// TwinCAT 3 PLC project Intecre_Events
// Title: Intecre.Events
// Company: Intecre Ltd
// Author: Mit Patel
// ProjectVersion: 0.1.1.2
// Description: V0.1.1.0 - Initial V0.1.1.1 - Create RPC Sink V0.1.1.2 - Separate Buffer and Sink Interfaces
// ProgramVersion: 3.1.4024.0
// libraries:
//   Intecre.Utilities, * (Intecre Ltd)
//   Tc2_EtherCAT, * (Beckhoff Automation GmbH)
//   Tc2_Standard, * (Beckhoff Automation GmbH)
//   Tc2_System, * (Beckhoff Automation GmbH)
//   Tc2_Utilities, * (Beckhoff Automation GmbH)
//   Tc3_JsonXml, * (Beckhoff Automation GmbH)
//   Intecre.File,newest,Intecre Ltd
// project tree:
//   Library/EventLogger/EventBuffers/ T_JsonEventBuffer.TcPOU (not stored)
//   Library/EventLogger/EventSinks/ T_RpcEventSink.TcPOU, FB_CsvFileEventSink.TcPOU
//   Library/EventLogger/Interfaces/ I_EventSink.TcIO, I_EventBuffer.TcIO, I_EventLogger.TcIO, I_Logger.TcIO (not stored), I_EventSeverityHandler.TcIO, I_EventSinkHandler.TcIO (not stored)
//   Library/Structs/ ST_EventMessageBuffer.TcDUT, ST_EventMessageBufferPool.TcDUT (not stored), ST_EventMessageParams.TcDUT (not stored), T_BufferString.TcDUT (not stored), T_MessageString.TcDUT
//   Library/EventLogger/Bases/ T_InstanceNameBase.TcPOU
//   Library/EventLogger/Functions/ F_GetLogSeverityFromTcEventSeverity.TcPOU
//   Library/EventLogger/ T_EventLogger.TcPOU, T_Logger.TcPOU (not stored)
//   Library/GVLs/ Events.TcGVL (not stored), EventsConfig.TcGVL
//   Library/Time/ FB_UnixTimestamp.TcPOU (not stored), I_TimeProvider.TcIO
//   Project Information/ F_GetCompany.TcPOU, F_GetTitle.TcPOU, F_GetVersion.TcPOU
//   Version/ Global_Version.TcGVL

// ---- Library/Structs/ST_EventMessageBuffer.TcDUT
{attribute 'pack_mode' := '0'}
TYPE ST_EventMessageBuffer :
STRUCT
 	bufferIndex : UINT := 0;
	availableForWriting : BOOL := TRUE;
  count : UINT := 0;
  timestampMs : ULINT;
  
  bufferSize : UDINT := EventsConfig.MAX_BUFFER_SIZE;
  dataSize : UDINT := 0;
END_STRUCT
END_TYPE

// ---- Library/Structs/T_MessageString.TcDUT
TYPE T_MessageString : STRING(EventsConfig.MAX_LOG_MESSAGE_SIZE); END_TYPE

// ---- Library/GVLs/EventsConfig.TcGVL
{attribute 'qualified_only'}
// Buffer Config
VAR_GLOBAL CONSTANT
  MAX_BUFFERS : UINT := 4;                    // Number of buffers.
  MAX_BUFFER_SIZE : UDINT := 65535;           // Max size in bytes of a buffer.
  CYCLE_BUFFERS : BOOL := TRUE;               // Overwrite buffers when all buffers are full.
  MAX_LOG_MESSAGE_SIZE : UINT := 512;         // Max length of log message.
  
  CSV_LOG_FILE_NAME : T_MaxString := 'logs';      // Name for CSV log files. Will have the date appended (e.g. logs_2024_05_26).
  CSV_LOG_FILE_PATH : T_MaxString := '/var/log/'; // The path for log files if using FB_CsvFileEventSink.
END_VAR

// Logs config
VAR_GLOBAL CONSTANT
  MAX_SINKS : UINT := 4; // Number of sinks.
END_VAR

// ---- Version/Global_Version.TcGVL
{attribute 'TcGenerated'}
{attribute 'no-analysis'}
{attribute 'linkalways'}
// This function has been automatically generated from the project information.
VAR_GLOBAL CONSTANT
	{attribute 'const_non_replaced'}
	stLibVersion_Intecre_Events : ST_LibVersion := (iMajor := 0, iMinor := 1, iBuild := 1, iRevision := 2, nFlags := 0, sVersion := '0.1.1.2');
END_VAR

// ---- Library/EventLogger/Interfaces/I_EventSink.TcIO
// Interface for consuming and exposing event logs for transmitting to an event receiver/ listener.
INTERFACE I_EventSink

// Adds an event to the sink for processing.
METHOD AddEvent
VAR_INPUT
  eventMessageParams : ST_EventMessageParams;
END_VAR
END_METHOD

// Gets events currently stored in the buffer and copies them to the resultString.
METHOD GetEvents : T_BufferString;
END_METHOD

// Initialises the sink including an I_TimeProvider for timestamping events.
METHOD Initialise
VAR_INPUT
	timeProvider : I_TimeProvider;
END_VAR
END_METHOD

END_INTERFACE

// ---- Library/EventLogger/Interfaces/I_EventBuffer.TcIO
// Interface for buffering event logs.
INTERFACE I_EventBuffer

// Adds an event to the buffer for later processing.
METHOD AddEvent
VAR_INPUT
  eventMessageParams : ST_EventMessageParams;
END_VAR
END_METHOD

// Gets events currently stored in the buffer and copies them to the resultString, returning the total length of bytes copied.
METHOD GetEvents : UDINT
VAR_INPUT
  resultString : REFERENCE TO T_BufferString;
END_VAR
END_METHOD

// Initialises the buffer including an I_TimeProvider for timestamping buffers and events.
METHOD Initialise
VAR_INPUT
	timeProvider : I_TimeProvider;
END_VAR
END_METHOD

END_INTERFACE

// ---- Library/EventLogger/Interfaces/I_EventLogger.TcIO
// Internal interface for general logging methods required by all loggers.
INTERFACE INTERNAL I_EventLogger

// Generic logging method.
METHOD INTERNAL LogEvent
VAR_IN_OUT CONSTANT
  message : T_MessageString; 
  sourceInstanceName : T_MaxString;
END_VAR

VAR_INPUT
  severity : TcEventSeverity;
END_VAR
END_METHOD

// Checks severity filters for whether the log message/ event should be logged.
METHOD INTERNAL ShouldLogEvent : BOOL
VAR_INPUT
  severity : TcEventSeverity;
END_VAR
END_METHOD

END_INTERFACE

// ---- Library/EventLogger/Interfaces/I_EventSeverityHandler.TcIO
// Interface for setting/ clearing local severity level.
INTERFACE I_EventSeverityHandler

// Clear the currently set local severity level.
METHOD ClearLocalSeverity
END_METHOD

// Get global severity level.
METHOD GetGlobalSeverity : TcEventSeverity
END_METHOD

// Get local severity level.
METHOD GetLocalSeverity : TcEventSeverity
END_METHOD

// Set a global severity level to filter logged events.
METHOD SetGlobalSeverity
VAR_INPUT
  severity : TcEventSeverity;
END_VAR
END_METHOD

// Set a local severity level to filter logged events. Ensure clear is called once local logging is complete.
METHOD SetLocalSeverity
VAR_INPUT
  severity : TcEventSeverity;
END_VAR
END_METHOD

END_INTERFACE

// ---- Library/Time/I_TimeProvider.TcIO
INTERFACE I_TimeProvider

PROPERTY TimestampMs : ULINT
GET
END_GET
END_PROPERTY

END_INTERFACE

// ---- Library/EventLogger/EventSinks/FB_CsvFileEventSink.TcPOU
// Event sink which writes log messages/ events to a CSV file. 
FUNCTION_BLOCK PUBLIC FB_CsvFileEventSink EXTENDS T_InstanceNameBase IMPLEMENTS I_EventSink
VAR
  isInitialised : BOOL := FALSE;
  
  csvFileWriter : T_CsvFileWriter;
  
  _timeProvider : I_TimeProvider := NULL;
  
  // Timeout timer to write messages in the T_CsvFileWriter's buffer after a timeout period.
  timeoutDuration : TIME := T#2S;         
  startTimer : BOOL := TRUE;
  timeoutTrigger : TON := (IN := startTimer, PT := timeoutDuration);
  
  task : T_Task;
  currentDateTime : T_MaxString;
  eventId : ULINT := 0;
END_VAR

VAR CONSTANT
  NULL : UDINT := 0;
END_VAR

// Adds an event to the sink for processing.
METHOD PUBLIC AddEvent
VAR_INPUT
  eventMessageParams : ST_EventMessageParams;
END_VAR
IF NOT isInitialised THEN
  F_LogWarning(CONCAT(InstanceName, ': Unable to AddEvent. Sink is uninitialised.'));
  RETURN;
END_IF

IF task.DateString <> currentDateTime THEN
  currentDateTime := task.DateString;
  csvFileWriter.SetFileParams(F_Concat3(EventsConfig.CSV_LOG_FILE_PATH, F_Concat3(EventsConfig.CSV_LOG_FILE_NAME, '_', currentDateTime), '.csv'), ASCI_COMMA);
END_IF

csvFileWriter.AddStringField(TO_STRING(eventId));
csvFileWriter.AddStringField(TO_STRING(_timeProvider.TimestampMs));
csvFileWriter.AddStringField(TO_STRING(eventMessageParams.Severity));
csvFileWriter.AddStringField(eventMessageParams.Source);
csvFileWriter.AddStringField(eventMessageParams.Message);

// Todo. Additional fields, unix timestamp, event id etc.

csvFileWriter.NewLine();
eventId := eventId + 1;
END_METHOD

METHOD PUBLIC CyclicLogic
IF NOT isInitialised THEN
  F_LogWarning(CONCAT(InstanceName, ': Unable to Execute. Sink is uninitialised.'));
  RETURN;
END_IF

csvFileWriter();

timeoutTrigger(IN := startTimer); // Restart timer on next cycle if triggered
IF timeoutTrigger.Q THEN
  timeoutTrigger(IN := FALSE);
  GetEvents();                    // Write data in the buffer.
END_IF
END_METHOD

// Gets events currently stored in the buffer and copies them to the resultString.
METHOD PUBLIC GetEvents : T_BufferString;
IF NOT isInitialised THEN
  F_LogWarning(CONCAT(InstanceName, ': Unable to GetEvents. Sink is uninitialised.'));
  RETURN;
END_IF

csvFileWriter.WriteToFile();
END_METHOD

// Initialises the buffer including an I_TimeProvider for timestamping buffers and events.
METHOD PUBLIC Initialise
VAR_INPUT
	timeProvider : I_TimeProvider;
END_VAR
_timeProvider := timeProvider;

IF _timeProvider = NULL THEN
  F_LogWarning(CONCAT(InstanceName, ': Unable to Initialise. _timeProvider is uninitialised.'));
  RETURN;
END_IF

isInitialised := TRUE;

currentDateTime := task.DateString;
csvFileWriter.SetFileOpenMode(TRUE);
csvFileWriter.SetFileParams(F_Concat3(EventsConfig.CSV_LOG_FILE_PATH, F_Concat3(EventsConfig.CSV_LOG_FILE_NAME, '_', currentDateTime), '.csv'), ASCI_COMMA);
END_METHOD

END_FUNCTION_BLOCK

// ---- Library/EventLogger/Bases/T_InstanceNameBase.TcPOU
{attribute 'reflection'} 
FUNCTION_BLOCK PUBLIC T_InstanceNameBase
VAR
  {attribute 'instance-path'} 
  {attribute 'noinit'} 
  name : T_MaxString;
  
  _instanceName : T_MaxString;
  isInstanceNameSet : BOOL := FALSE;
END_VAR

PROPERTY FINAL InstanceName : T_MaxString; // returns the fully scoped variable name
GET
IF NOT isInstanceNameSet THEN
   setInstanceName();
END_IF

InstanceName := _instanceName;
END_GET
END_PROPERTY

METHOD PRIVATE SetInstanceName
VAR
	charsToDeleteFromPath : INT;
END_VAR
//Remove Solution_Name
charsToDeleteFromPath := FIND(name, '.');
_instanceName := DELETE(name, charsToDeleteFromPath, 1);
//Remove ProjectName
charsToDeleteFromPath := FIND(_instanceName, '.');
//gives us just "FirstDeclaredPOU.etc.etc..." from above.
_instanceName := DELETE(_instanceName, charsToDeleteFromPath, 1);
END_METHOD

END_FUNCTION_BLOCK

// ---- Library/EventLogger/EventSinks/T_RpcEventSink.TcPOU
// Event sink which buffers log messages/ events ready for polling via RPC calls to 'GetEvents'; a method of the I_EventSink interface. 
FUNCTION_BLOCK PUBLIC T_RpcEventSink EXTENDS T_InstanceNameBase IMPLEMENTS I_EventSink
VAR
  jsonBuffer : T_JsonEventBuffer;
END_VAR

// Adds an event to the sink for processing.
METHOD PUBLIC AddEvent
VAR_INPUT
  eventMessageParams : ST_EventMessageParams;
END_VAR
jsonBuffer.AddEvent(eventMessageParams);
END_METHOD

// Gets events currently stored in the buffer and copies them to the resultString.
{attribute 'TcRpcEnable'}
METHOD PUBLIC GetEvents : T_BufferString;
jsonBuffer.GetEvents(GetEvents);
END_METHOD

// Initialises the buffer including an I_TimeProvider for timestamping buffers and events.
METHOD PUBLIC Initialise
VAR_INPUT
	timeProvider : I_TimeProvider;
END_VAR
jsonBuffer.Initialise(timeProvider);
END_METHOD

END_FUNCTION_BLOCK

// ---- Library/EventLogger/Functions/F_GetLogSeverityFromTcEventSeverity.TcPOU
// Conversion helper to convert from TcEventSeverity to Intecre.Utilities E_LogSeverity.
FUNCTION INTERNAL F_GetLogSeverityFromTcEventSeverity : E_LogSeverity
VAR_INPUT
  severity : TcEventSeverity;
END_VAR

CASE severity OF

  TcEventSeverity.Verbose   : F_GetLogSeverityFromTcEventSeverity := E_LogSeverity.Debug;
  TcEventSeverity.Info      : F_GetLogSeverityFromTcEventSeverity := E_Logseverity.Info;
  TcEventSeverity.Warning   : F_GetLogSeverityFromTcEventSeverity := E_Logseverity.Warning;
  TcEventSeverity.Error     : F_GetLogSeverityFromTcEventSeverity := E_Logseverity.Error;
  TcEventSeverity.Critical  : F_GetLogSeverityFromTcEventSeverity := E_Logseverity.Error;

END_CASE

END_FUNCTION

// ---- Library/EventLogger/T_EventLogger.TcPOU
// Internal logger which allows adding/ clearing sinks to be processed, in addition to receiving log events and forwarding them to sinks.
FUNCTION_BLOCK INTERNAL T_EventLogger EXTENDS T_InstanceNameBase IMPLEMENTS I_EventLogger, I_Logger, I_EventSinkHandler, I_EventSeverityHandler;
VAR
  eventSinks : ARRAY[1..EventsConfig.MAX_SINKS] OF I_EventSink;
  eventSinksCount : UINT := 0;
  
  globalSeverity : TcEventSeverity; // Global log filter.
  localSeverity : TcEventSeverity;
  useLocalSeverity : BOOL;
END_VAR

VAR CONSTANT
  NULL : UDINT := 0;
END_VAR

// Adds a sink to the sink handler and returns TRUE if successful.
METHOD PUBLIC AddSink : BOOL
VAR_INPUT
	sink	: I_EventSink;
END_VAR
IF eventSinksCount + 1 > EventsConfig.MAX_SINKS THEN
  F_LogWarning(CONCAT(InstanceName, ': Unable to add sink. Maximum number of event sinks reached'));
  RETURN;
END_IF

eventSinksCount := eventSinksCount + 1;
eventSinks[eventSinksCount] := sink;
AddSink := TRUE;
END_METHOD

// Clear the currently set local severity level.
METHOD PUBLIC ClearLocalSeverity
useLocalSeverity := FALSE;
END_METHOD

// Clears all sinks currently being handled by the sink handler.
METHOD PUBLIC ClearSinks
VAR
  iSink : UINT := 0;
END_VAR
IF eventSinksCount > 0 AND eventSinksCount <= EventsConfig.MAX_SINKS THEN
  FOR iSink := 1 TO eventSinksCount DO
    eventSinks[iSink] := NULL;
  END_FOR
END_IF

eventSinksCount := 0;
END_METHOD

// Get global severity level.
METHOD GetGlobalSeverity : TcEventSeverity
GetGlobalSeverity := globalSeverity;
END_METHOD

// Get local severity level.
METHOD GetLocalSeverity : TcEventSeverity
GetLocalSeverity := localSeverity;
END_METHOD

METHOD PUBLIC LogCritical
VAR_INPUT
  message : T_MessageString; 
END_VAR

VAR
  localInstanceName : T_MaxString;
END_VAR
localInstanceName := InstanceName;
LogEvent(message := message, sourceInstanceName := localInstanceName, severity := TcEventSeverity.Critical);
END_METHOD

METHOD PUBLIC LogError
VAR_INPUT
  message : T_MessageString; 
END_VAR

VAR
  localInstanceName : T_MaxString;
END_VAR
localInstanceName := InstanceName;
LogEvent(message := message, sourceInstanceName := localInstanceName, severity := TcEventSeverity.Error);
END_METHOD

METHOD INTERNAL LogEvent
VAR_IN_OUT CONSTANT
  message : T_MessageString; 
  sourceInstanceName : T_MaxString;
END_VAR

VAR_INPUT
  severity : TcEventSeverity;
END_VAR

VAR
  iSink : UINT := 0;
  adsLogSeverity : E_LogSeverity;
  eventMessageParams : ST_EventMessageParams;
END_VAR
IF NOT ShouldLogEvent(severity) THEN
  RETURN;
END_IF

eventMessageParams.Message := message;
eventMessageParams.Severity := severity;
eventMessageParams.Source := sourceInstanceName;

IF eventSinksCount > 0 AND eventSinksCount <= EventsConfig.MAX_SINKS THEN
  FOR iSink := 1 TO eventSinksCount DO
    IF eventSinks[iSink] <> NULL THEN
      eventSinks[iSink].AddEvent(eventMessageParams);
    ELSE
      F_LogWarning(CONCAT(InstanceName, ': Unable to LogEvent. Sink is uninitialised.'));
    END_IF
  END_FOR
END_IF

adsLogSeverity := F_GetLogSeverityFromTcEventSeverity(severity);
F_Logger(
  LogSeverity := adsLogSeverity,
  Message := F_Concat3(sourceInstanceName, ': ', message)
);
END_METHOD

METHOD PUBLIC LogInfo
VAR_INPUT
  message : T_MessageString; 
END_VAR

VAR
  localInstanceName : T_MaxString;
END_VAR
localInstanceName := InstanceName;
LogEvent(message := message, sourceInstanceName := localInstanceName, severity := TcEventSeverity.Info);
END_METHOD

METHOD PUBLIC LogVerbose
VAR_INPUT
  message : T_MessageString; 
END_VAR

VAR
  localInstanceName : T_MaxString;
END_VAR
localInstanceName := InstanceName;
LogEvent(message := message, sourceInstanceName := localInstanceName, severity := TcEventSeverity.Verbose);
END_METHOD

METHOD PUBLIC LogWarning
VAR_INPUT
  message : T_MessageString; 
END_VAR

VAR
  localInstanceName : T_MaxString;
END_VAR
localInstanceName := InstanceName;
LogEvent(message := message, sourceInstanceName := localInstanceName, severity := TcEventSeverity.Warning);
END_METHOD

// Set a global severity level to filter logged events.
METHOD PUBLIC SetGlobalSeverity
VAR_INPUT
	severity	: TcEventSeverity;
END_VAR
globalSeverity := severity;
END_METHOD

// Set a local severity level to filter logged events. Ensure clear is called once local logging is complete.
METHOD PUBLIC SetLocalSeverity
VAR_INPUT
	severity	: TcEventSeverity;
END_VAR
localSeverity := severity;
useLocalSeverity := TRUE;
END_METHOD

METHOD INTERNAL ShouldLogEvent : BOOL
VAR_INPUT
  severity : TcEventSeverity;
END_VAR
IF useLocalSeverity THEN
  ShouldLogEvent := severity >= localSeverity;  
ELSE
  ShouldLogEvent := severity >= globalSeverity;
END_IF
END_METHOD

END_FUNCTION_BLOCK

// ---- Project Information/F_GetCompany.TcPOU
// This function has been automatically generated from the project information.
{attribute 'signature_flag' := '1073741824'}
{attribute 'TcGenerated'}
{attribute 'no-analysis'}
FUNCTION F_GetCompany : WSTRING
VAR_INPUT
	
END_VAR

F_GetCompany := "Intecre Ltd";

END_FUNCTION

// ---- Project Information/F_GetTitle.TcPOU
// This function has been automatically generated from the project information.
{attribute 'signature_flag' := '1073741824'}
{attribute 'TcGenerated'}
{attribute 'no-analysis'}
FUNCTION F_GetTitle : WSTRING
VAR_INPUT
	
END_VAR

F_GetTitle := "Intecre.Events";

END_FUNCTION

// ---- Project Information/F_GetVersion.TcPOU
// This function has been automatically generated from the project information.
{attribute 'signature_flag' := '1073741824'}
{attribute 'TcGenerated'}
{attribute 'no-analysis'}
FUNCTION F_GetVersion : ST_LibVersion
VAR_INPUT
	
END_VAR

F_GetVersion.iMajor := 0;
F_GetVersion.iMinor := 1;
F_GetVersion.iBuild := 1;
F_GetVersion.iRevision := 2;
F_GetVersion.sVersion := '0.1.1.2';
F_GetVersion.nFlags := 0;

END_FUNCTION
